FUNCTION_BLOCK FINAL FBAdd
VAR_INPUT
	a:WORD;
	b:WORD;
END_VAR
VAR_OUTPUT
	c:word;
END_VAR
VAR
END_VAR

c:=a+b;
c:=a*b;

ACTION ACT:

END_ACTION

METHOD PUBLIC METH : BOOL
VAR_INPUT
END_VAR
END_METHOD

METHOD PRIVATE METH_1 : BOOL
VAR_INPUT
END_VAR
END_METHOD

PROPERTY PUBLIC Prop : INT
GET
END_GET
SET
END_SET
END_PROPERTY

END_FUNCTION_BLOCK

(* stored: Version 1.1.0.1, ProductVersion 3.1.4024.12
   POU FBAdd: Id {29fb77bd-f8c0-45c3-9487-63510db585b9}, SpecialFunc None
   Action ACT: Id {bee8ad85-aa8d-4494-9081-15a1ea7f8e8b}
   Method METH: Id {29786db5-ab6c-4fac-a0bf-0a76773a00e8}
   Method METH_1: Id {60deb40c-6aea-478c-b679-814979b6539d}
   Property Prop: Id {ea3b9da3-2cfb-4e08-81e8-de3b707d97e5}
   Get Get: Id {2c202a84-21f1-4f29-ba36-37125ab48062}
   Set Set: Id {0caf9444-e951-41a3-a4cb-321e8e0a0f5e} *)
